PROGRAM EXAMPLE_MAIN
VAR
    _context : ExampleCylinderContext;
END_VAR

_context.Run();

END_PROGRAM

(* stored: Version 1.1.0.1, ProductVersion 3.1.4024.10
   POU EXAMPLE_MAIN: Id {2c5d3f02-495c-0bc3-10fa-11136d9736d0}, SpecialFunc None *)
